// Mitsubishi GX Works2 project: GX W2 L5 Ex 2 DK C   PLC: FX3G

// task Task_01 (event TRUE, interval 0, priority 31): POU_01

PROGRAM POU_01
IF X001 THEN
D2 := 5;   (* When X1 is turned On, the Constant 5 is moved into Data Register D2 *)
END_IF;
IF X002 THEN
D2 := D2 + 1;   (* When X2 is turned On, D2 will increment based on the Scan Cycle by the value of 1 (Ensure X1 is OFF) *)
END_IF;
END_PROGRAM
